Omron CX-Programmer project NewProject (CX-Programmer 9.50)

# PLC TUBESOI: CP1H XA

## Global symbols (name address type ; comment)
0 CHANNEL  ; DIGITAL DISPLAY
0.00 BOOL  ; PB START
0.01 BOOL  ; PB STOP
0.02 BOOL  ; VISION SENSOR 1
0.03 BOOL  ; VISION SENSOR 2
0.04 BOOL  ; VISION SENSOR 3
0.05 BOOL  ; VISION SENSOR 4
0.06 BOOL  ; LID CLAMPED
0.07 BOOL  ; LID AT PLACE
100.00 BOOL  ; L HIJAU
100.01 BOOL  ; L MERAH
100.02 BOOL  ; CONVEYOR 1 KANAN
100.03 BOOL  ; CONVEYOR 2 KIRI
100.04 BOOL  ; CONVEYOR 3 KANAN
100.05 BOOL  ; CONVEYOR 4 KIRI
100.06 BOOL  ; PIVOT ARM SORTER 1
100.07 BOOL  ; PIVOT ARM SORTER 2
101.00 BOOL  ; PIVOT ARM SORTER 1 BELT +
101.01 BOOL  ; PIVOT ARM SORTER 2 BELT +
101.02 BOOL  ; MOVE X
101.03 BOOL  ; MOVE Z
101.04 BOOL  ; GRAB
101.05 BOOL  ; CLAMP LID
101.06 BOOL  ; CLAMP BASE
101.07 BOOL  ; POS RAISE BASE
102.00 BOOL  ; POS RAISE LID GATE
102.01 BOOL  ; POS RAISE BASE GATE
102.02 BOOL  ; PIVOT ARM SORTER 3
102.03 BOOL  ; PIVOT ARM SORTER 3 BELT +
102.04 BOOL  ; BUZZER EMERGENCY
102.05 BOOL  ; L KUNING
102.06 BOOL  ; STACK MERAH
102.07 BOOL  ; STACK HIJAU
103.00 BOOL  ; STACK KUNING
103.01 BOOL  ; BLUE LID DISPLAY
1.00 BOOL  ; BASE AT PLACE
1.01 BOOL  ; LID GATE SENSOR
1.02 BOOL  ; BASE GATE SENSOR
1.03 BOOL  ; LID BLUE GOOD SENSOR
1.04 BOOL  ; LID GREEN GOOD SENSOR
1.05 BOOL  ; BASE BLUE GOOD
1.06 BOOL  ; BASE GREEN GOOD
1.07 BOOL  ; SORTING COLOUR BLUE
2.00 BOOL  ; K UTAMA
2.03 BOOL  ; LOCK GOOD PART LID
2.04 BOOL  ; LOCK GOOD PART BASE
2.05 BOOL  ; KONTAK SENSOR COLOUR
2.06 BOOL  ; E STOP
3.01 BOOL  ; EMERGENCY STOP
T0000 BOOL  ; TIMER PIVOT KANAN
T0001 BOOL  ; TIMER PIVOT KIRI

## Program NewProgram1 (cyclic task 0)

### Section Section1

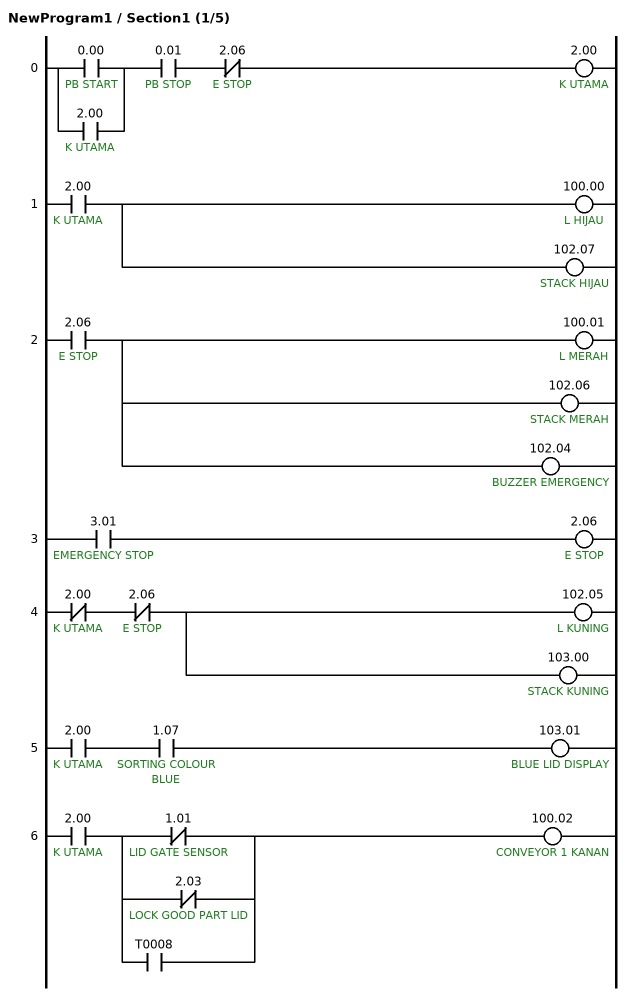
; rung 0
LD 0.00  ; PB START
OR 2.00  ; K UTAMA
AND 0.01  ; PB STOP
ANDNOT 2.06  ; E STOP
OUT 2.00  ; K UTAMA
; rung 1
LD 2.00  ; K UTAMA
OUT 100.00  ; L HIJAU
OUT 102.07  ; STACK HIJAU
; rung 2
LD 2.06  ; E STOP
OUT 100.01  ; L MERAH
OUT 102.06  ; STACK MERAH
OUT 102.04  ; BUZZER EMERGENCY
; rung 3
LD 3.01  ; EMERGENCY STOP
OUT 2.06  ; E STOP
; rung 4
LDNOT 2.00  ; K UTAMA
ANDNOT 2.06  ; E STOP
OUT 102.05  ; L KUNING
OUT 103.00  ; STACK KUNING
; rung 5
LD 2.00  ; K UTAMA
AND 1.07  ; SORTING COLOUR BLUE
OUT 103.01  ; BLUE LID DISPLAY
; rung 6
LD 2.00  ; K UTAMA
LDNOT 1.01  ; LID GATE SENSOR
ORNOT 2.03  ; LOCK GOOD PART LID
OR T0008
ANDLD
OUT 100.02  ; CONVEYOR 1 KANAN

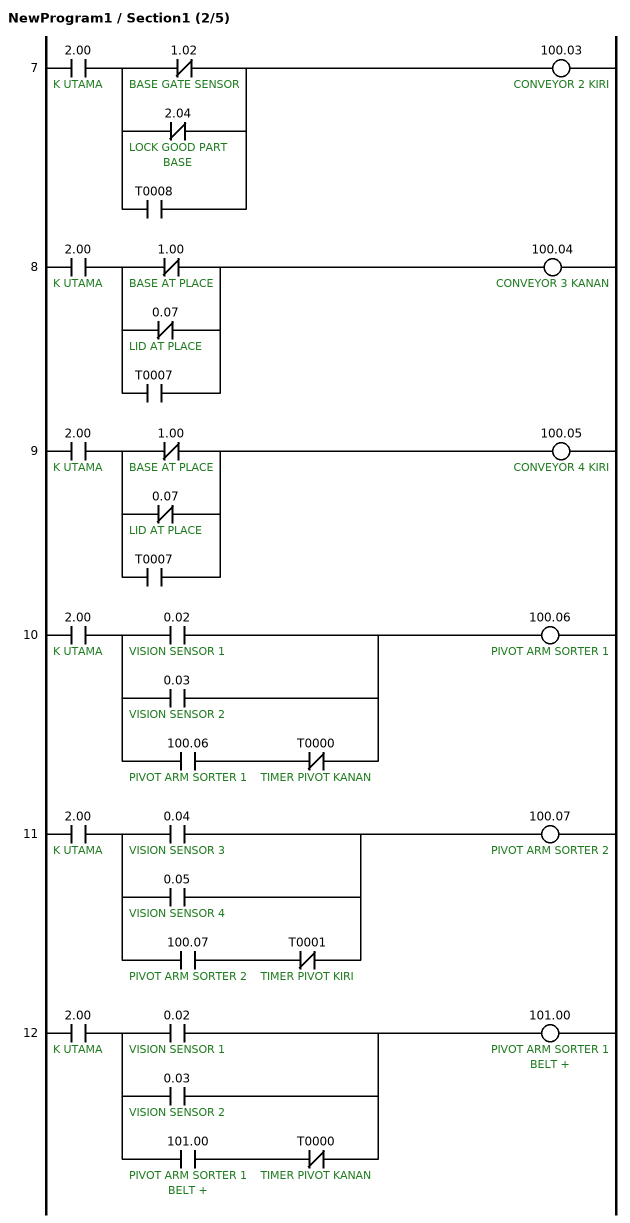
; rung 7
LD 2.00  ; K UTAMA
LDNOT 1.02  ; BASE GATE SENSOR
ORNOT 2.04  ; LOCK GOOD PART BASE
OR T0008
ANDLD
OUT 100.03  ; CONVEYOR 2 KIRI
; rung 8
LD 2.00  ; K UTAMA
LDNOT 1.00  ; BASE AT PLACE
ORNOT 0.07  ; LID AT PLACE
OR T0007
ANDLD
OUT 100.04  ; CONVEYOR 3 KANAN
; rung 9
LD 2.00  ; K UTAMA
LDNOT 1.00  ; BASE AT PLACE
ORNOT 0.07  ; LID AT PLACE
OR T0007
ANDLD
OUT 100.05  ; CONVEYOR 4 KIRI
; rung 10
LD 2.00  ; K UTAMA
LD 0.02  ; VISION SENSOR 1
OR 0.03  ; VISION SENSOR 2
LD 100.06  ; PIVOT ARM SORTER 1
ANDNOT T0000  ; TIMER PIVOT KANAN
ORLD
ANDLD
OUT 100.06  ; PIVOT ARM SORTER 1
; rung 11
LD 2.00  ; K UTAMA
LD 0.04  ; VISION SENSOR 3
OR 0.05  ; VISION SENSOR 4
LD 100.07  ; PIVOT ARM SORTER 2
ANDNOT T0001  ; TIMER PIVOT KIRI
ORLD
ANDLD
OUT 100.07  ; PIVOT ARM SORTER 2
; rung 12
LD 2.00  ; K UTAMA
LD 0.02  ; VISION SENSOR 1
OR 0.03  ; VISION SENSOR 2
LD 101.00  ; PIVOT ARM SORTER 1 BELT +
ANDNOT T0000  ; TIMER PIVOT KANAN
ORLD
ANDLD
OUT 101.00  ; PIVOT ARM SORTER 1 BELT +

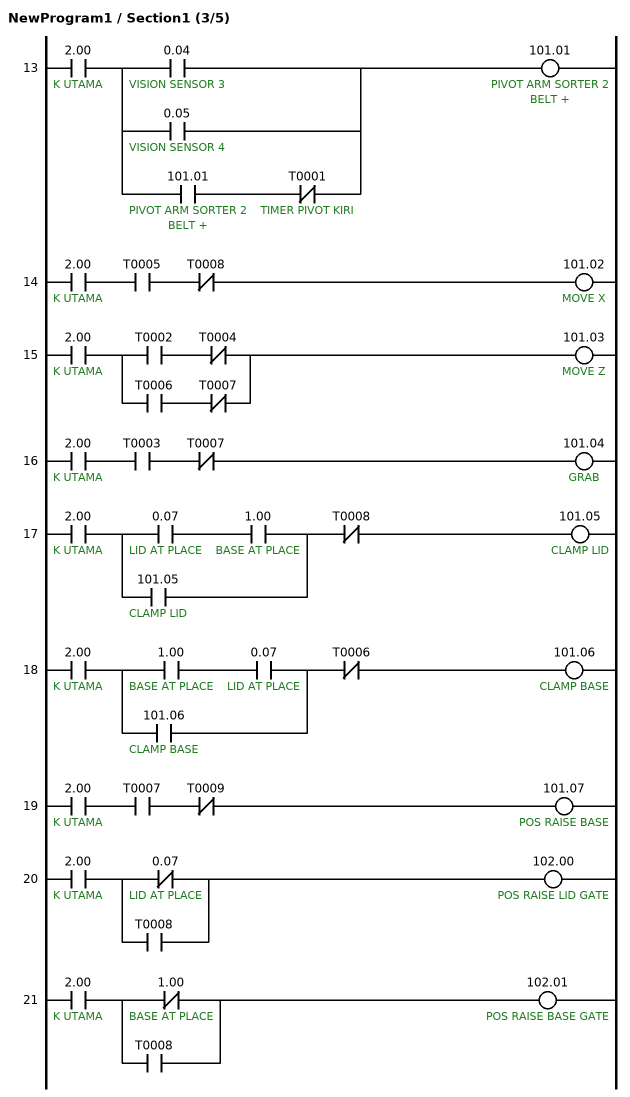
; rung 13
LD 2.00  ; K UTAMA
LD 0.04  ; VISION SENSOR 3
OR 0.05  ; VISION SENSOR 4
LD 101.01  ; PIVOT ARM SORTER 2 BELT +
ANDNOT T0001  ; TIMER PIVOT KIRI
ORLD
ANDLD
OUT 101.01  ; PIVOT ARM SORTER 2 BELT +
; rung 14
LD 2.00  ; K UTAMA
AND T0005
ANDNOT T0008
OUT 101.02  ; MOVE X
; rung 15
LD 2.00  ; K UTAMA
LD T0002
ANDNOT T0004
LD T0006
ANDNOT T0007
ORLD
ANDLD
OUT 101.03  ; MOVE Z
; rung 16
LD 2.00  ; K UTAMA
AND T0003
ANDNOT T0007
OUT 101.04  ; GRAB
; rung 17
LD 2.00  ; K UTAMA
LD 0.07  ; LID AT PLACE
AND 1.00  ; BASE AT PLACE
OR 101.05  ; CLAMP LID
ANDLD
ANDNOT T0008
OUT 101.05  ; CLAMP LID
; rung 18
LD 2.00  ; K UTAMA
LD 1.00  ; BASE AT PLACE
AND 0.07  ; LID AT PLACE
OR 101.06  ; CLAMP BASE
ANDLD
ANDNOT T0006
OUT 101.06  ; CLAMP BASE
; rung 19
LD 2.00  ; K UTAMA
AND T0007
ANDNOT T0009
OUT 101.07  ; POS RAISE BASE
; rung 20
LD 2.00  ; K UTAMA
LDNOT 0.07  ; LID AT PLACE
OR T0008
ANDLD
OUT 102.00  ; POS RAISE LID GATE
; rung 21
LD 2.00  ; K UTAMA
LDNOT 1.00  ; BASE AT PLACE
OR T0008
ANDLD
OUT 102.01  ; POS RAISE BASE GATE

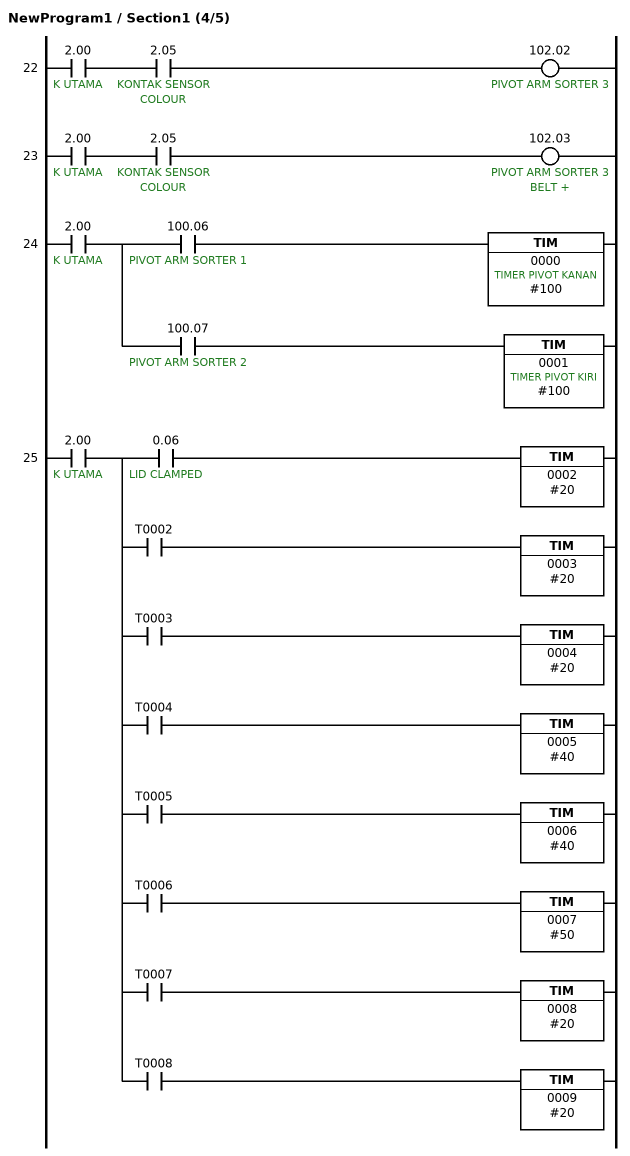
; rung 22
LD 2.00  ; K UTAMA
AND 2.05  ; KONTAK SENSOR COLOUR
OUT 102.02  ; PIVOT ARM SORTER 3
; rung 23
LD 2.00  ; K UTAMA
AND 2.05  ; KONTAK SENSOR COLOUR
OUT 102.03  ; PIVOT ARM SORTER 3 BELT +
; rung 24
LD 2.00  ; K UTAMA
OUT TR0
AND 100.06  ; PIVOT ARM SORTER 1
TIM 0000 #100  ; TIMER PIVOT KANAN
LD TR0
AND 100.07  ; PIVOT ARM SORTER 2
TIM 0001 #100  ; TIMER PIVOT KIRI
; rung 25
LD 2.00  ; K UTAMA
OUT TR0
AND 0.06  ; LID CLAMPED
TIM 0002 #20
LD TR0
AND T0002
TIM 0003 #20
LD TR0
AND T0003
TIM 0004 #20
LD TR0
AND T0004
TIM 0005 #40
LD TR0
AND T0005
TIM 0006 #40
LD TR0
AND T0006
TIM 0007 #50
LD TR0
AND T0007
TIM 0008 #20
LD TR0
AND T0008
TIM 0009 #20

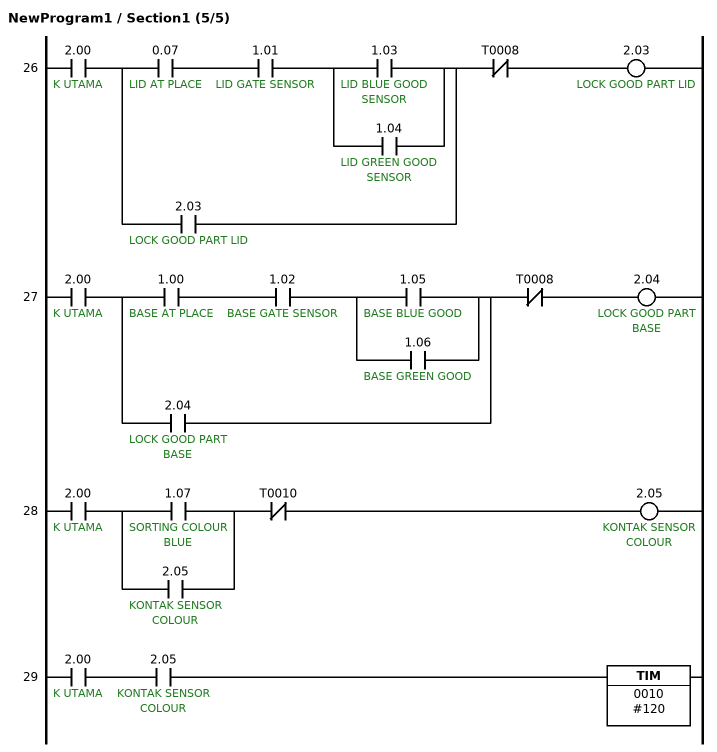
; rung 26
LD 2.00  ; K UTAMA
LD 0.07  ; LID AT PLACE
AND 1.01  ; LID GATE SENSOR
LD 1.03  ; LID BLUE GOOD SENSOR
OR 1.04  ; LID GREEN GOOD SENSOR
ANDLD
OR 2.03  ; LOCK GOOD PART LID
ANDLD
ANDNOT T0008
OUT 2.03  ; LOCK GOOD PART LID
; rung 27
LD 2.00  ; K UTAMA
LD 1.00  ; BASE AT PLACE
AND 1.02  ; BASE GATE SENSOR
LD 1.05  ; BASE BLUE GOOD
OR 1.06  ; BASE GREEN GOOD
ANDLD
OR 2.04  ; LOCK GOOD PART BASE
ANDLD
ANDNOT T0008
OUT 2.04  ; LOCK GOOD PART BASE
; rung 28
LD 2.00  ; K UTAMA
LD 1.07  ; SORTING COLOUR BLUE
OR 2.05  ; KONTAK SENSOR COLOUR
ANDLD
ANDNOT T0010
OUT 2.05  ; KONTAK SENSOR COLOUR
; rung 29
LD 2.00  ; K UTAMA
AND 2.05  ; KONTAK SENSOR COLOUR
TIM 0010 #120

### Section END
; rung 0
END(001)